// Mitsubishi GX Works2 project: PLC-Servo 실습 과제 4   PLC: Q03UDV

PROGRAM MAIN
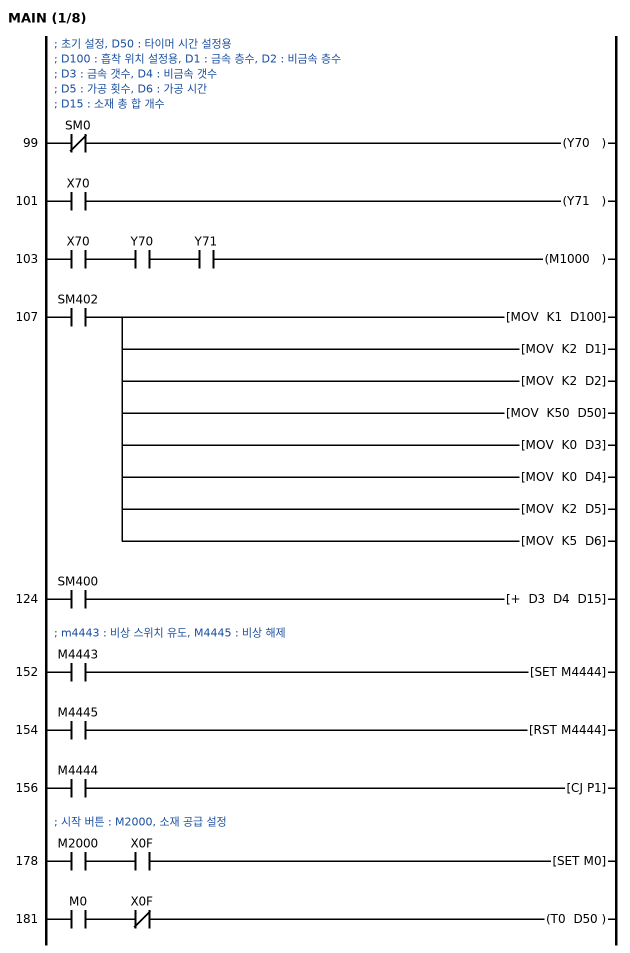
; 초기 설정, D50 : 타이머 시간 설정용
; D100 : 흡착 위치 설정용, D1 : 금속 층수, D2 : 비금속 층수
; D3 : 금속 갯수, D4 : 비금속 갯수
; D5 : 가공 횟수, D6 : 가공 시간
; D15 : 소재 총 합 개수
99    LDI     SM0
      OUT     Y70
101   LD      X70
      OUT     Y71
103   LD      X70
      AND     Y70
      AND     Y71
      OUT     M1000
107   LD      SM402
      MOV     K1 D100
      MOV     K2 D1
      MOV     K2 D2
      MOV     K50 D50
      MOV     K0 D3
      MOV     K0 D4
      MOV     K2 D5
      MOV     K5 D6
124   LD      SM400
      +       D3 D4 D15
; m4443 : 비상 스위치 유도, M4445 : 비상 해제
152   LD      M4443
      SET     M4444
154   LD      M4445
      RST     M4444
156   LD      M4444
      CJ      P1
; 시작 버튼 : M2000, 소재 공급 설정
178   LD      M2000
      AND     X0F
      SET     M0
181   LD      M0
      ANI     X0F
      OUT     T0 D50
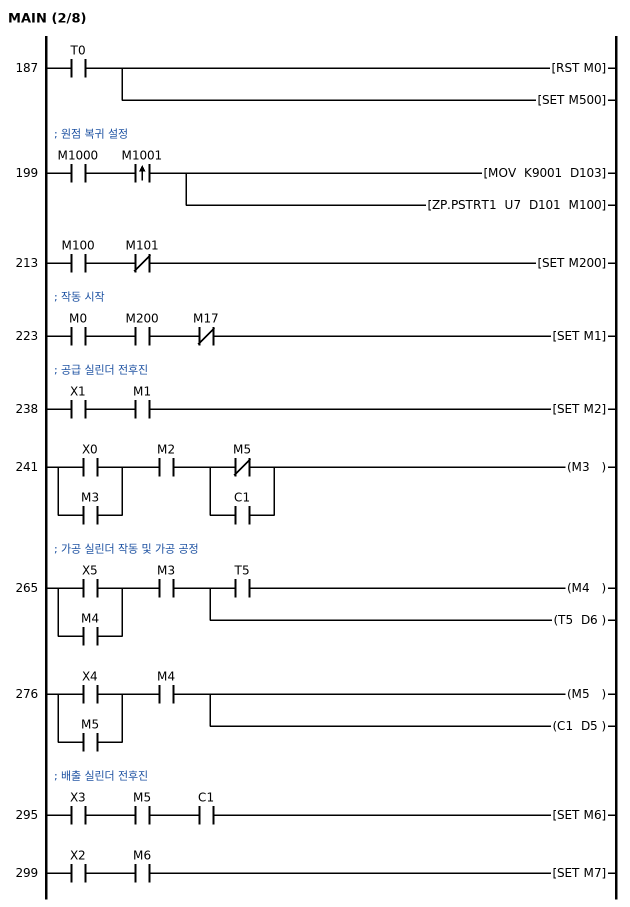
187   LD      T0
      RST     M0
      SET     M500
; 원점 복귀 설정
199   LD      M1000
      ANDP    M1001
      MOV     K9001 D103
      ZP.PSTRT1 U7 D101 M100
213   LD      M100
      ANI     M101
      SET     M200
; 작동 시작
223   LD      M0
      AND     M200
      ANI     M17
      SET     M1
; 공급 실린더 전후진
238   LD      X1
      AND     M1
      SET     M2
241   LD      X0
      OR      M3
      AND     M2
      LDI     M5
      OR      C1
      ANB
      OUT     M3
; 가공 실린더 작동 및 가공 공정
265   LD      X5
      OR      M4
      AND     M3
      MPS
      AND     T5
      OUT     M4
      MPP
      OUT     T5 D6
276   LD      X4
      OR      M5
      AND     M4
      OUT     M5
      OUT     C1 D5
; 배출 실린더 전후진
295   LD      X3
      AND     M5
      AND     C1
      SET     M6
299   LD      X2
      AND     M6
      SET     M7
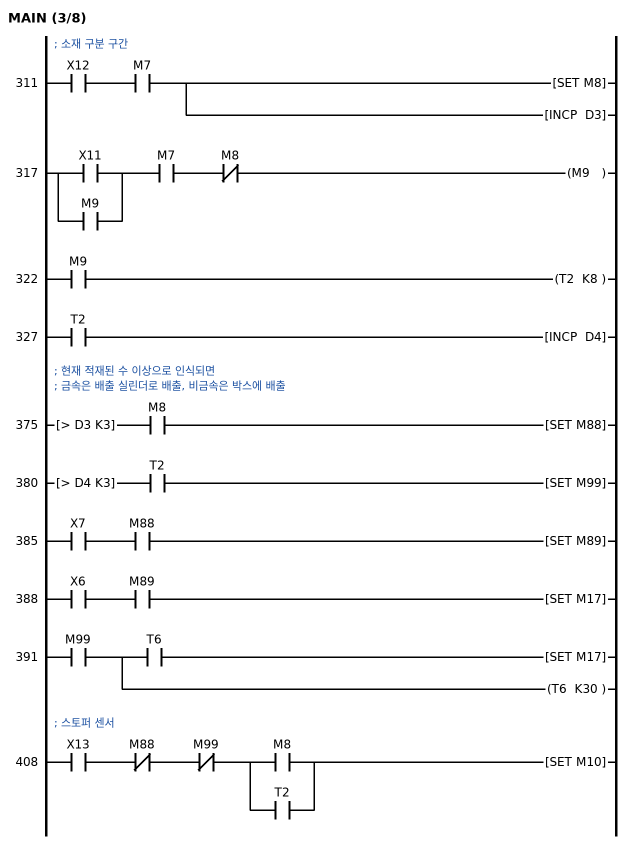
; 소재 구분 구간
311   LD      X12
      AND     M7
      SET     M8
      INCP    D3
317   LD      X11
      OR      M9
      AND     M7
      ANI     M8
      OUT     M9
322   LD      M9
      OUT     T2 K8
327   LD      T2
      INCP    D4
; 현재 적재된 수 이상으로 인식되면
; 금속은 배출 실린더로 배출, 비금속은 박스에 배출
375   LD>     D3 K3
      AND     M8
      SET     M88
380   LD>     D4 K3
      AND     T2
      SET     M99
385   LD      X7
      AND     M88
      SET     M89
388   LD      X6
      AND     M89
      SET     M17
391   LD      M99
      MPS
      AND     T6
      SET     M17
      MPP
      OUT     T6 K30
; 스토퍼 센서
408   LD      X13
      ANI     M88
      ANI     M99
      LD      M8
      OR      T2
      ANB
      SET     M10
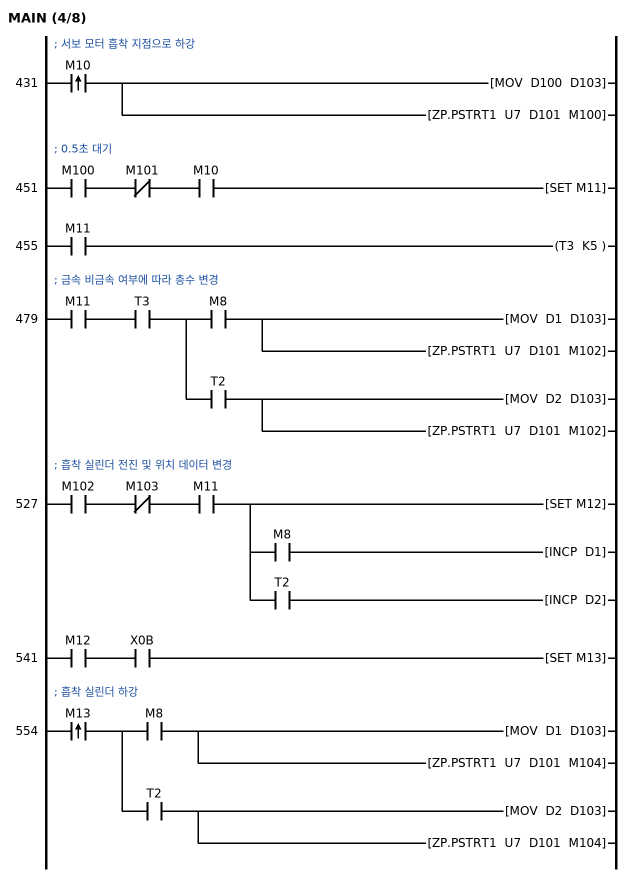
; 서보 모터 흡착 지점으로 하강
431   LDP     M10
      MOV     D100 D103
      ZP.PSTRT1 U7 D101 M100
; 0.5초 대기
451   LD      M100
      ANI     M101
      AND     M10
      SET     M11
455   LD      M11
      OUT     T3 K5
; 금속 비금속 여부에 따라 층수 변경
479   LD      M11
      AND     T3
      MPS
      AND     M8
      MOV     D1 D103
      ZP.PSTRT1 U7 D101 M102
      MPP
      AND     T2
      MOV     D2 D103
      ZP.PSTRT1 U7 D101 M102
; 흡착 실린더 전진 및 위치 데이터 변경
527   LD      M102
      ANI     M103
      AND     M11
      SET     M12
      MPS
      AND     M8
      INCP    D1
      MPP
      AND     T2
      INCP    D2
541   LD      M12
      AND     X0B
      SET     M13
; 흡착 실린더 하강
554   LDP     M13
      MPS
      AND     M8
      MOV     D1 D103
      ZP.PSTRT1 U7 D101 M104
      MPP
      AND     T2
      MOV     D2 D103
      ZP.PSTRT1 U7 D101 M104
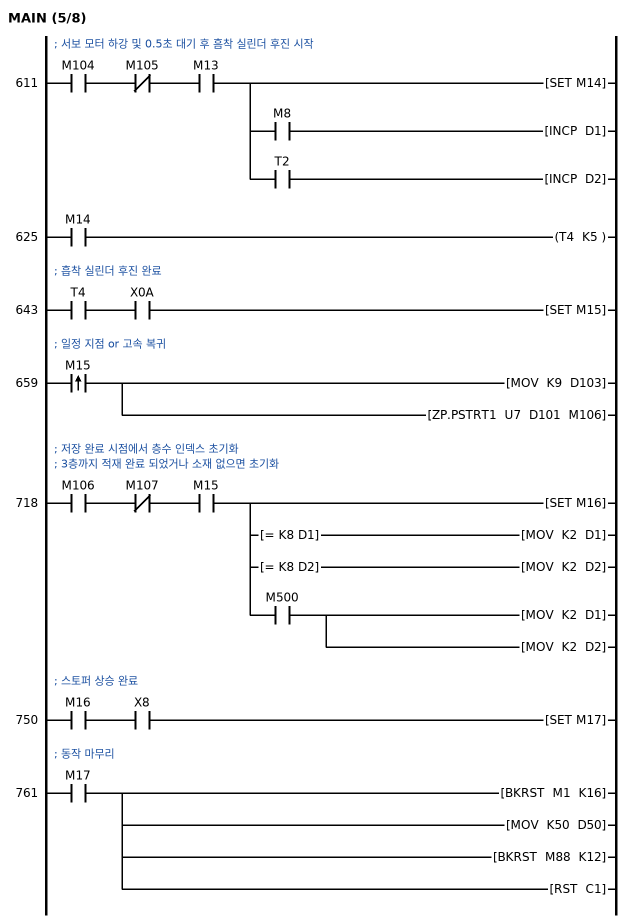
; 서보 모터 하강 및 0.5초 대기 후 흠착 실린더 후진 시작
611   LD      M104
      ANI     M105
      AND     M13
      SET     M14
      MPS
      AND     M8
      INCP    D1
      MPP
      AND     T2
      INCP    D2
625   LD      M14
      OUT     T4 K5
; 흡착 실린더 후진 완료
643   LD      T4
      AND     X0A
      SET     M15
; 일정 지점 or 고속 복귀
659   LDP     M15
      MOV     K9 D103
      ZP.PSTRT1 U7 D101 M106
; 저장 완료 시점에서 층수 인덱스 초기화
; 3층까지 적재 완료 되었거나 소재 없으면 초기화
718   LD      M106
      ANI     M107
      AND     M15
      SET     M16
      MPS
      AND=    K8 D1
      MOV     K2 D1
      MRD
      AND=    K8 D2
      MOV     K2 D2
      MPP
      AND     M500
      MOV     K2 D1
      MOV     K2 D2
; 스토퍼 상승 완료
750   LD      M16
      AND     X8
      SET     M17
; 동작 마무리
761   LD      M17
      BKRST   M1 K16
      MOV     K50 D50
      BKRST   M88 K12
      RST     C1
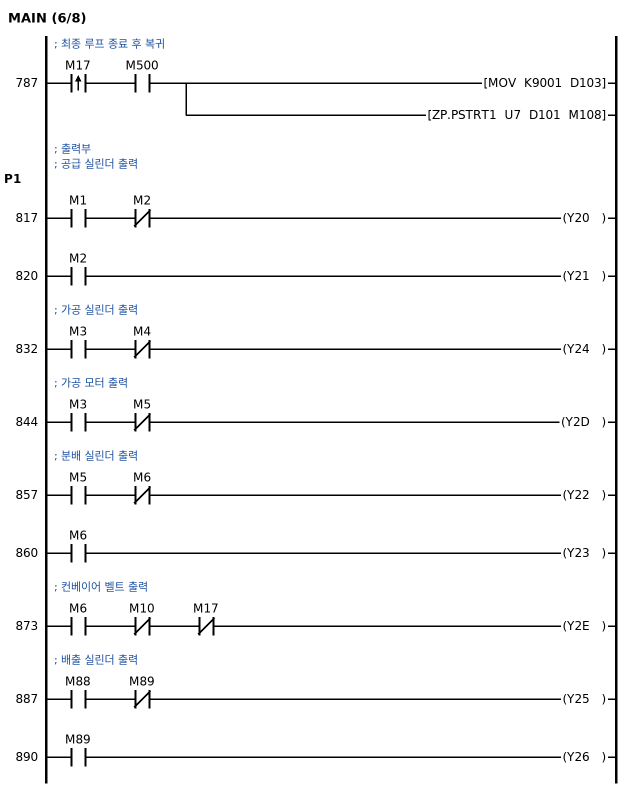
; 최종 루프 종료 후 복귀
787   LDP     M17
      AND     M500
      MOV     K9001 D103
      ZP.PSTRT1 U7 D101 M108
; 출력부
; 공급 실린더 출력
      P1
817   LD      M1
      ANI     M2
      OUT     Y20
820   LD      M2
      OUT     Y21
; 가공 실린더 출력
832   LD      M3
      ANI     M4
      OUT     Y24
; 가공 모터 출력
844   LD      M3
      ANI     M5
      OUT     Y2D
; 분배 실린더 출력
857   LD      M5
      ANI     M6
      OUT     Y22
860   LD      M6
      OUT     Y23
; 컨베이어 벨트 출력
873   LD      M6
      ANI     M10
      ANI     M17
      OUT     Y2E
; 배출 실린더 출력
887   LD      M88
      ANI     M89
      OUT     Y25
890   LD      M89
      OUT     Y26
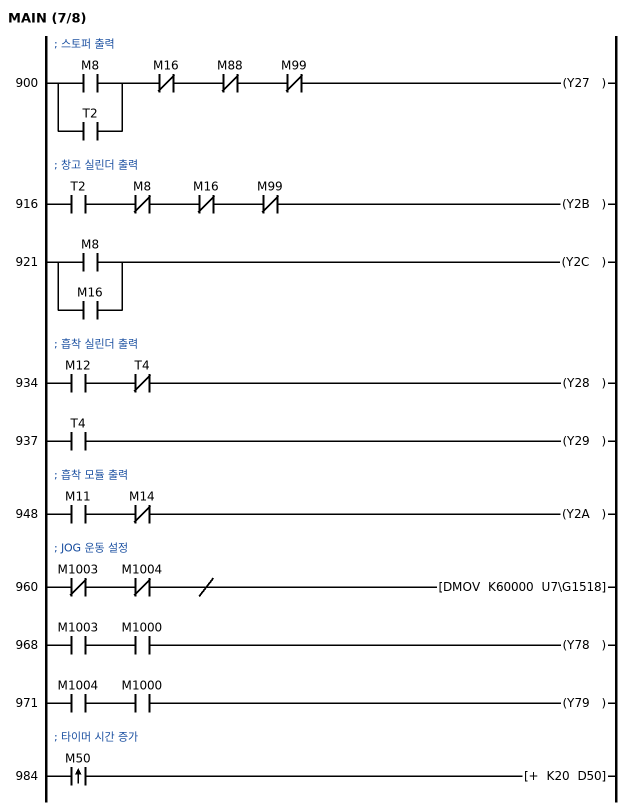
; 스토퍼 출력
900   LD      M8
      OR      T2
      ANI     M16
      ANI     M88
      ANI     M99
      OUT     Y27
; 창고 실린더 출력
916   LD      T2
      ANI     M8
      ANI     M16
      ANI     M99
      OUT     Y2B
921   LD      M8
      OR      M16
      OUT     Y2C
; 흡착 실린더 출력
934   LD      M12
      ANI     T4
      OUT     Y28
937   LD      T4
      OUT     Y29
; 흡착 모듈 출력
948   LD      M11
      ANI     M14
      OUT     Y2A
; JOG 운동 설정
960   LDI     M1003
      ANI     M1004
      INV
      DMOV    K60000 U7\G1518
968   LD      M1003
      AND     M1000
      OUT     Y78
971   LD      M1004
      AND     M1000
      OUT     Y79
; 타이머 시간 증가
984   LDP     M50
      +       K20 D50
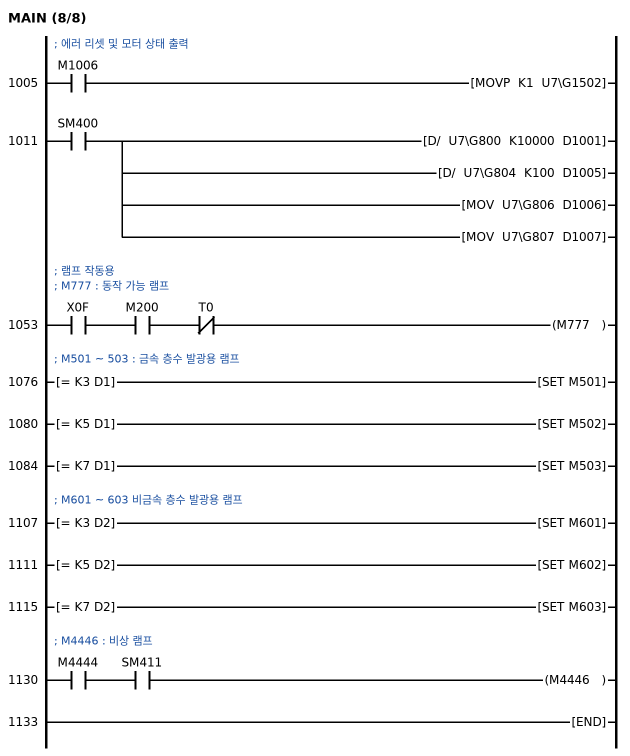
; 에러 리셋 및 모터 상태 출력
1005  LD      M1006
      MOVP    K1 U7\G1502
1011  LD      SM400
      D/      U7\G800 K10000 D1001
      D/      U7\G804 K100 D1005
      MOV     U7\G806 D1006
      MOV     U7\G807 D1007
; 램프 작동용
; M777 : 동작 가능 램프
1053  LD      X0F
      AND     M200
      ANI     T0
      OUT     M777
; M501 ~ 503 : 금속 층수 발광용 램프
1076  LD=     K3 D1
      SET     M501
1080  LD=     K5 D1
      SET     M502
1084  LD=     K7 D1
      SET     M503
; M601 ~ 603 비금속 층수 발광용 램프
1107  LD=     K3 D2
      SET     M601
1111  LD=     K5 D2
      SET     M602
1115  LD=     K7 D2
      SET     M603
; M4446 : 비상 램프
1130  LD      M4444
      AND     SM411
      OUT     M4446
1133  END
END_PROGRAM
